FUNCTION_BLOCK Conveyor 
VAR_INPUT
END_VAR

VAR_OUTPUT
	bStart  : BOOL;
END_VAR
VAR
	fbStart : BoolOut;
END_VAR

bStart := fbStart.getValue;

PROPERTY getStart : I_StepCondition
GET
getStart := fbStart;
END_GET
END_PROPERTY

METHOD Off : BOOL
VAR_INPUT
END_VAR
fbStart.setValue := FALSE;
END_METHOD

METHOD On : BOOL
VAR_INPUT
END_VAR
fbStart.setValue := TRUE;
END_METHOD

END_FUNCTION_BLOCK

(* stored: Version 1.1.0.1, ProductVersion 3.1.4024.2
   POU Conveyor: Id {e1227bcb-2673-40d9-b87d-ebff2f2762dc}, SpecialFunc None
   Property getStart: Id {4f7a1143-3cc3-4e3a-830c-c1cee2508c6f}
   Get Get: Id {8d1c48dd-37d7-4fae-86fd-9449fb147fce}
   Method Off: Id {ad914a28-e08e-4d14-9ea5-dbfbd01d37d4}
   Method On: Id {ea37b98a-aa0e-4a0e-bc89-47a3ebe7a0e6} *)
